{attribute 'call_after_init'}
FUNCTION_BLOCK FINAL RealParam EXTENDS BaseParam
VAR_INPUT
END_VAR
VAR_OUTPUT
	value: REAL;
END_VAR
VAR
	
END_VAR

METHOD Change_Param
VAR_INPUT
	value	: STRING;
END_VAR
THIS^.value := STRING_TO_REAL(value);
_display := REAL_TO_STRING(THIS^.value);
END_METHOD

METHOD Quick_Change
VAR_INPUT
	value: REAL;
END_VAR
THIS^.value := value;
_display := REAL_TO_STRING(THIS^.value);
END_METHOD

END_FUNCTION_BLOCK

(* stored: Version 1.1.0.1, ProductVersion 3.1.4024.12
   POU RealParam: Id {bde2d684-dcab-4662-9463-a66ca463423c}, SpecialFunc None
   Method Change_Param: Id {db107ac4-93d8-4a09-9702-afdbda642683}
   Method Quick_Change: Id {59e493e8-5b5b-4e98-8ea9-05bb57eb2e2d} *)
